// TIA Portal V18 export
FUNCTION "mot_set_speed_by_target_multiturn_util1" : Void   // FC23, FBD
{ S7_Optimized_Access := 'TRUE' }
VERSION : 0.1
// stored: AutoNumber true, IsIECCheckEnabled false, SetENOAutomatically false, UDAEnableTagReadback false
   VAR_INPUT
      target : Real;
      delta : Real;
      pos : Real;
   END_VAR
   VAR_OUTPUT
      distance : Real;
      target_plus_delta : Real;
   END_VAR
BEGIN

REGION Network 2 (SCL)
   #target_plus_delta := #target + #delta
   ;
END_REGION

REGION Network 3 (SCL)
   #distance:= ABS(#target_plus_delta - #pos);
END_REGION
END_FUNCTION
